//==================================================================================================
//								RJM Maszyny sp. z o.o.
//									13.05.2022
//
//	Obsługa przycisku podświetlanego
//	v1.0	|| TC v 3.1.4024.22		|| - pierwsza wersja
//==================================================================================================
FUNCTION_BLOCK FB_Przycisk_NC_Podswietlany EXTENDS FB_Przycisk_NC
VAR
	bLampka							AT %Q*	: BOOL;
	
END_VAR

//==================================================================================================
//								RJM Maszyny sp. z o.o.
//									13.05.2022
//
//	Włączenie podświetlenia przycisku
//	v1.0	|| TC v 3.1.4024.22		|| - pierwsza wersja
//==================================================================================================
METHOD WlaczPodswietlenie
VAR_INPUT
END_VAR
bLampka										:= TRUE;
END_METHOD

//==================================================================================================
//								RJM Maszyny sp. z o.o.
//									13.05.2022
//
//	Wyłączenie podświetlenia przycisku
//	v1.0	|| TC v 3.1.4024.22		|| - pierwsza wersja
//==================================================================================================
METHOD WylaczPodswietlenie
VAR_INPUT
END_VAR
bLampka										:= FALSE;
END_METHOD

END_FUNCTION_BLOCK

(* stored: Version 1.1.0.1, ProductVersion 3.1.4024.11
   POU FB_Przycisk_NC_Podswietlany: Id {a4d35e9d-2bf9-419f-86bb-904560e64ad0}, SpecialFunc None
   Method WlaczPodswietlenie: Id {81282c3e-9e01-4171-b730-1a76e35e675e}
   Method WylaczPodswietlenie: Id {3e73d794-83dc-4f34-8239-07b6c11c7978} *)
